// TIA Portal V17 export
// export: Created 2022-03-11T11:27:36.1676076Z, ExportSetting WithDefaults, DisplayName Totally Integrated Automation Portal, DisplayVersion V17, DisplayName TIA Portal Openness, DisplayVersion V17, DisplayName TIA Portal Version Control Interface, DisplayVersion V17, DisplayName STEP 7 Professional, DisplayVersion V17, DisplayName STEP 7 Safety, DisplayVersion V17, DisplayName WinCC Advanced, DisplayVersion V17
FUNCTION "Inputs_1" : Void   // FC2, FBD
{ S7_Optimized_Access := 'TRUE' }
VERSION : 0.1
// stored: AutoNumber true, IsIECCheckEnabled false, SetENOAutomatically false, UDAEnableTagReadback false
   VAR_INPUT
      input0 : Bool;
      input1 : Bool;
      input2 : Bool;
      input3 : Bool;
   END_VAR
   VAR_OUTPUT
      output0 : Bool;
      output1 : Bool;
      output2 : Bool;
      output3 : Bool;
   END_VAR
BEGIN
END_FUNCTION
